FUNCTION_BLOCK PrintStatus (* goFB_ignore *)
  (* Standard: 61499-2 *)
  (* Version 0.1, 2017-00-16, hpea485, UOA *)
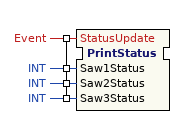
  EVENT_INPUT
    StatusUpdate WITH Saw1Status, Saw2Status, Saw3Status;
  END_EVENT
  VAR_INPUT
    Saw1Status : INT;
    Saw2Status : INT;
    Saw3Status : INT;
  END_VAR
  EC_STATES
    Start;
  END_STATES
END_FUNCTION_BLOCK
